(* PLC project Untitled1, Beckhoff Automation GmbH TF6420 Database Server Query Analyser 1.0.0.0 *)
(* stored: creationDateTime 2022-01-14T14:12:36, modificationDateTime 2022-01-14T14:12:36 *)

TYPE ST_SelectStructIMU : STRUCT
  datetime : STRING(255);
  trailer_id_lead : LINT;
  trailer_id_rear : LINT;
  pitch_lead : REAL;
  roll_lead : REAL;
  ax_lead : REAL;
  ay_lead : REAL;
  az_lead : REAL;
  pitch_rear : REAL;
  roll_rear : REAL;
  ax_rear : REAL;
  ay_rear : REAL;
  az_rear : REAL;
END_STRUCT;
END_TYPE
